FUNCTION F_PadWith : STRING
VAR_INPUT
	in_Int:INT;
	in_NumOfBytes:INT;
	in_PadWith:STRING;
END_VAR
VAR
	i:INT;
	TempString:STRING;
END_VAR

TempString := '';

FOR i := 1 TO in_NumOfBytes - LEN(INT_TO_STRING(in_INT)) DO
	TempString := CONCAT(TempString, in_PadWith);
END_FOR

F_PadWith := CONCAT(TempString, INT_TO_STRING(in_INT));

END_FUNCTION

(* stored: Version 1.1.0.1, ProductVersion 3.1.4024.5
   POU F_PadWith: Id {48352928-08b4-43fd-85f0-1f7fbe59f1ba}, SpecialFunc None *)
